(* CODESYS project BagFeedMotorIMove.Calculate_entry.xml

Project tree, tasks and I/O mapping:
*)

// Calculate_entry
ACTION Calculate_entry:
_Destination := Count + Steps;
END_ACTION
